// TIA Portal project "Automacao" (V16)
// Vorlageprojekt für das Buch mit Zielsystem S7-1200

(* hardware
DEVICE "S7-1200-Station_1"  S7-1200 Station
   slot 0: "Baugruppenträger_0"  Rack  V1.0
   slot 1: "PLC_1"  CPU 1211C DC/DC/DC  6ES7 211-1AE40-0XB0  V4.1
*)

// ===== PLC "PLC_1"  CPU 1211C DC/DC/DC =====

VAR_GLOBAL   // PLC tag table "Standard-Variablentabelle"
   "Start" AT %I0.1 : Bool;
   "Stop" AT %I0.3 : Bool;
   "Entry_conveyor" AT %Q0.0 : Bool;
   "Exit_conveyor" AT %Q0.2 : Bool;
   "Sort_1_turn" AT %Q0.3 : Bool;
   "Sort_1_belt" AT %Q0.4 : Bool;
   "Sort_2_turn" AT %Q0.5 : Bool;
   "Sort_2_belt" AT %Q0.6 : Bool;
   "Sort_3_turn" AT %Q0.7 : Bool;
   "Sort_3_belt" AT %Q1.0 : Bool;
   "At_exit" AT %I0.0 : Bool;
   "Vision_sensor" AT %ID30 : DInt;
   "active_separation_1" AT %M0.1 : Bool;
   "active_separation_2" AT %M0.2 : Bool;
   "active_separation_3" AT %M0.3 : Bool;
   "Tag_1" AT %M2.0 : Bool;
   "Tag_2" AT %M2.1 : Bool;
END_VAR

FUNCTION "MHJ-PLC-Lab-Function-S71200" : Void   // FC9000, SCL
{ S7_Optimized_Access := 'TRUE' }
VERSION : 0.1
   VAR_TEMP
      rdTimeReturn : Int;
      outputTime : DTL;
      SyncVal : Byte;
      forVal : Int;
      forVal_2 : Int;
      Value : Byte;
   END_VAR
   VAR CONSTANT
      CompVal : Byte := 16#34;
      Value_01 : Byte := 16#11;
      Value_01_DW : DWord := 16#A165_D992;
      Value_02_DW : DWord := 16#58BE_4401;
   END_VAR
BEGIN

   #Value:=PEEK(area := 16#82,
        dbNumber := 0,
        byteOffset := 511);
   #Value := #Value + 1;

   POKE(area := 16#82,
        dbNumber := 0,
        byteOffset := 511,
        value := #Value);

   POKE(area:=16#81,
        dbNumber:=0,
        byteOffset:=1016,
        value:=#Value_01_DW);
   POKE(area := 16#81,
        dbNumber := 0,
        byteOffset := 1020,
        value := #Value_02_DW);

   POKE(area := 16#81,
        dbNumber := 0,
        byteOffset := 511,
        value := B#16#00);

   FOR #forVal := 0 TO 120 DO
       FOR #forVal_2:=0 TO 10 DO
           #rdTimeReturn:=RD_SYS_T(#outputTime);
           #rdTimeReturn := WR_SYS_T(#outputTime);
           #rdTimeReturn := RD_SYS_T(#outputTime);
           #rdTimeReturn := WR_SYS_T(#outputTime);
       END_FOR;
       #SyncVal:= PEEK(area := 16#81,
                      dbNumber := 0,
                      byteOffset := 511);
       IF #SyncVal = #CompVal THEN
          GOTO M_1;
       END_IF;
   END_FOR;
   RETURN;

   M_1:
   POKE(area := 16#81,
        dbNumber := 0,
        byteOffset := 511,
        value := B#16#0);
END_FUNCTION

ORGANIZATION_BLOCK "Main"   // OB1, LAD, ProgramCycle
TITLE = "Main Program Sweep (Cycle)"
{ S7_Optimized_Access := 'TRUE' }
VERSION : 0.1
   VAR_INPUT
      Initial_Call : Bool;   // Initial call of this OB
      Remanence : Bool;   // =True, if remanent data are available
   END_VAR
   VAR_TEMP   // added for the SCL form of the ladder/FBD networks
      _w1 : Bool;
      _w2 : Bool;
   END_VAR
BEGIN

REGION Network 1: Konnektierungsbaustein für PLC-Lab
   // Im Netzwerk 1 wird der Konnektierungsbaustein für PLC-Lab aufgerufen.
   // Dieser Aufruf darf nicht entfernt werden!
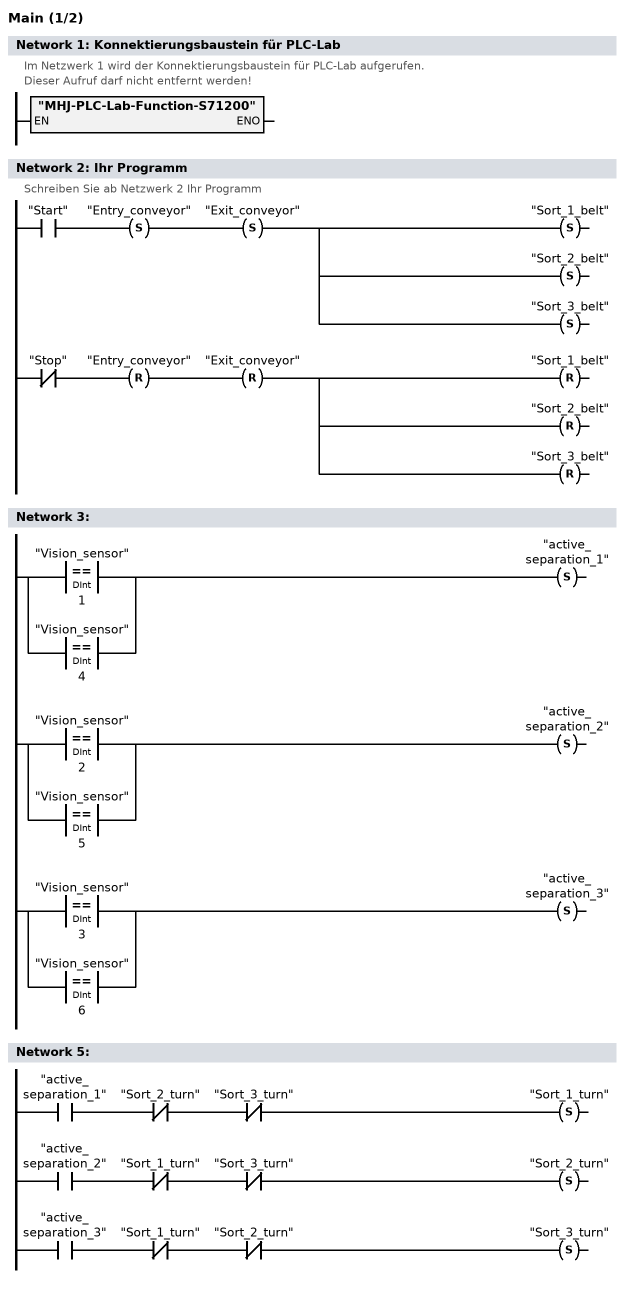
   RUNG wire#powerrail
      "MHJ-PLC-Lab-Function-S71200"()
   END_RUNG
   // the same network as SCL:
   "MHJ-PLC-Lab-Function-S71200"();
END_REGION

REGION Network 2: Ihr Programm
   // Schreiben Sie ab Netzwerk 2 Ihr Programm
   RUNG wire#powerrail
      Contact( "Start" )
      S_Coil( "Entry_conveyor" )
      S_Coil( "Exit_conveyor" )
      wire#w1
      S_Coil( "Sort_1_belt" )
   END_RUNG
   RUNG wire#w1
      S_Coil( "Sort_2_belt" )
   END_RUNG
   RUNG wire#w1
      S_Coil( "Sort_3_belt" )
   END_RUNG
   RUNG wire#powerrail
      I_Contact( "Stop" )
      R_Coil( "Entry_conveyor" )
      R_Coil( "Exit_conveyor" )
      wire#w2
      R_Coil( "Sort_1_belt" )
   END_RUNG
   RUNG wire#w2
      R_Coil( "Sort_2_belt" )
   END_RUNG
   RUNG wire#w2
      R_Coil( "Sort_3_belt" )
   END_RUNG
   // the same network as SCL:
   IF "Start" THEN
       "Entry_conveyor" := TRUE;
       "Exit_conveyor" := TRUE;
       "Sort_1_belt" := TRUE;
       "Sort_2_belt" := TRUE;
       "Sort_3_belt" := TRUE;
   END_IF;
   IF NOT "Stop" THEN
       "Entry_conveyor" := FALSE;
       "Exit_conveyor" := FALSE;
       "Sort_1_belt" := FALSE;
       "Sort_2_belt" := FALSE;
       "Sort_3_belt" := FALSE;
   END_IF;
END_REGION

REGION Network 3
   RUNG wire#powerrail
      { S7_Templates := "SrcType := DInt" } EQ_Contact(in1 := "Vision_sensor", in2 := 1)
      wire#w1
      S_Coil( "active_separation_1" )
   END_RUNG
   RUNG wire#powerrail
      { S7_Templates := "SrcType := DInt" } EQ_Contact(in1 := "Vision_sensor", in2 := 4)
   END_RUNG wire#w1
   RUNG wire#powerrail
      { S7_Templates := "SrcType := DInt" } EQ_Contact(in1 := "Vision_sensor", in2 := 2)
      wire#w2
      S_Coil( "active_separation_2" )
   END_RUNG
   RUNG wire#powerrail
      { S7_Templates := "SrcType := DInt" } EQ_Contact(in1 := "Vision_sensor", in2 := 5)
   END_RUNG wire#w2
   RUNG wire#powerrail
      { S7_Templates := "SrcType := DInt" } EQ_Contact(in1 := "Vision_sensor", in2 := 3)
      wire#w3
      S_Coil( "active_separation_3" )
   END_RUNG
   RUNG wire#powerrail
      { S7_Templates := "SrcType := DInt" } EQ_Contact(in1 := "Vision_sensor", in2 := 6)
   END_RUNG wire#w3
   // the same network as SCL:
   IF ("Vision_sensor" = 1) OR ("Vision_sensor" = 4) THEN "active_separation_1" := TRUE; END_IF;
   IF ("Vision_sensor" = 2) OR ("Vision_sensor" = 5) THEN "active_separation_2" := TRUE; END_IF;
   IF ("Vision_sensor" = 3) OR ("Vision_sensor" = 6) THEN "active_separation_3" := TRUE; END_IF;
END_REGION

REGION Network 5
   RUNG wire#powerrail
      Contact( "active_separation_1" )
      I_Contact( "Sort_2_turn" )
      I_Contact( "Sort_3_turn" )
      S_Coil( "Sort_1_turn" )
   END_RUNG
   RUNG wire#powerrail
      Contact( "active_separation_2" )
      I_Contact( "Sort_1_turn" )
      I_Contact( "Sort_3_turn" )
      S_Coil( "Sort_2_turn" )
   END_RUNG
   RUNG wire#powerrail
      Contact( "active_separation_3" )
      I_Contact( "Sort_1_turn" )
      I_Contact( "Sort_2_turn" )
      S_Coil( "Sort_3_turn" )
   END_RUNG
   // the same network as SCL:
   IF "active_separation_1" AND NOT "Sort_2_turn" AND NOT "Sort_3_turn" THEN "Sort_1_turn" := TRUE; END_IF;
   IF "active_separation_2" AND NOT "Sort_1_turn" AND NOT "Sort_3_turn" THEN "Sort_2_turn" := TRUE; END_IF;
   IF "active_separation_3" AND NOT "Sort_1_turn" AND NOT "Sort_2_turn" THEN "Sort_3_turn" := TRUE; END_IF;
END_REGION

REGION Network 6
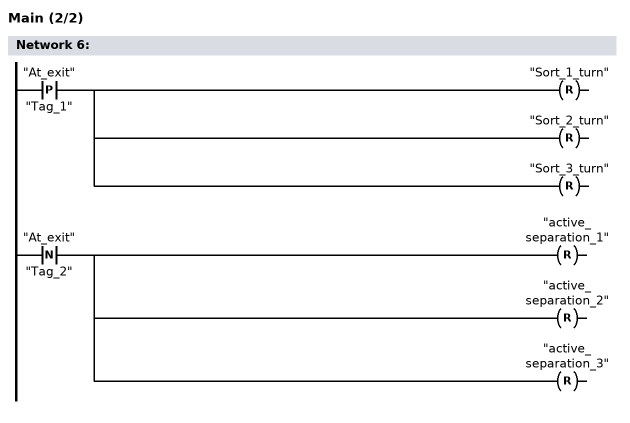
   RUNG wire#powerrail
      P_Contact(operand := "At_exit", bit := "Tag_1")
      wire#w1
      R_Coil( "Sort_1_turn" )
   END_RUNG
   RUNG wire#w1
      R_Coil( "Sort_2_turn" )
   END_RUNG
   RUNG wire#w1
      R_Coil( "Sort_3_turn" )
   END_RUNG
   RUNG wire#powerrail
      N_Contact(operand := "At_exit", bit := "Tag_2")
      wire#w2
      R_Coil( "active_separation_1" )
   END_RUNG
   RUNG wire#w2
      R_Coil( "active_separation_2" )
   END_RUNG
   RUNG wire#w2
      R_Coil( "active_separation_3" )
   END_RUNG
   // the same network as SCL:
   #_w1 := "At_exit" AND NOT "Tag_1";   // rising edge of "At_exit"
   "Tag_1" := "At_exit";
   IF #_w1 THEN
       "Sort_1_turn" := FALSE;
       "Sort_2_turn" := FALSE;
       "Sort_3_turn" := FALSE;
   END_IF;
   #_w2 := NOT "At_exit" AND "Tag_2";   // falling edge of "At_exit"
   "Tag_2" := "At_exit";
   IF #_w2 THEN
       "active_separation_1" := FALSE;
       "active_separation_2" := FALSE;
       "active_separation_3" := FALSE;
   END_IF;
END_REGION
END_ORGANIZATION_BLOCK